(* IEC 61131-3 sources: vertical-injection-machine-docs/docs/IM_SYS_PRG/Code/面板管理/面板公用, 7 files *)

(* ---- PanelTypes.st ---- *)
(*
  PanelTypes.st
  功能：
  1. 定义面板管理层统一使用的按键点位结构和综合按键结构。
  2. 统一收口“面板排序号 + 按键值 + 按键灯”三类信息，避免键值与灯值分散绑定。
  3. 为 `FB_MK110`、`FB_MK116`、`FB_MK150` 提供稳定的数据边界。

  说明：
  1. `uiPanelOrder` 由具体面板功能块按各自型号写入，`0` 表示当前面板未安装该逻辑键位。
  2. `bValue` 由面板输入解码逻辑回写，表示当前逻辑键是否被按下。
  3. `bLamp` 由上层控制逻辑写入，表示当前逻辑键对应的灯是否需要点亮。
*)

TYPE ST_PanelButton :
STRUCT
    uiPanelOrder: UINT;     // 当前逻辑键在当前面板型号中的排序号；`0` 表示该面板型号不提供此键位。
    bValue: BOOL;           // 当前逻辑键输入值；由面板功能块根据输入字和排序号解码后回写。
    bLamp: BOOL;            // 当前逻辑键灯输出请求；由上层写入，再由面板功能块按排序号编码到输出字。
END_STRUCT
END_TYPE

TYPE ST_PanelButtons :
STRUCT
    stManual: ST_PanelButton;            // 手动键综合点位，统一收口其排序号、键值和灯值。
    stSemiautomatic: ST_PanelButton;     // 半自动键综合点位，统一收口其排序号、键值和灯值。
    stAutomatic: ST_PanelButton;         // 全自动键综合点位，统一收口其排序号、键值和灯值。
    stAdjustMold: ST_PanelButton;        // 调模键综合点位，统一收口其排序号、键值和灯值。
    stHeat: ST_PanelButton;              // 电热键综合点位，统一收口其排序号、键值和灯值。
    stMotor: ST_PanelButton;             // 马达键综合点位，统一收口其排序号、键值和灯值。
    stMoldOpen: ST_PanelButton;          // 开模键综合点位，统一收口其排序号、键值和灯值。
    stMoldClose: ST_PanelButton;         // 锁模键综合点位，统一收口其排序号、键值和灯值。
    stMaterialMelt: ST_PanelButton;      // 储料键综合点位，统一收口其排序号、键值和灯值。
    stCleanMaterial: ST_PanelButton;     // 清料键综合点位，统一收口其排序号、键值和灯值。
    stJetLube: ST_PanelButton;           // 润滑键综合点位，统一收口其排序号、键值和灯值。
    stInjFwd: ST_PanelButton;            // 射出键综合点位，统一收口其排序号、键值和灯值。
    stInjBwd: ST_PanelButton;            // 射退键综合点位，统一收口其排序号、键值和灯值。
    stPressRise: ST_PanelButton;         // 压力加键综合点位，统一收口其排序号、键值和灯值。
    stPressFall: ST_PanelButton;         // 压力减键综合点位，统一收口其排序号、键值和灯值。
    stEjectorFwd: ST_PanelButton;        // 托模进键综合点位，统一收口其排序号、键值和灯值。
    stEjectorBwd: ST_PanelButton;        // 托模退键综合点位，统一收口其排序号、键值和灯值。
    stMultiEjector: ST_PanelButton;      // 多次托模键综合点位，统一收口其排序号、键值和灯值。
    stBlow: ST_PanelButton;              // 吹气键综合点位，统一收口其排序号、键值和灯值。
    stInjUnitFwd: ST_PanelButton;        // 座进键综合点位，统一收口其排序号、键值和灯值。
    stInjUnitBwd: ST_PanelButton;        // 座退键综合点位，统一收口其排序号、键值和灯值。
    stLockFwd: ST_PanelButton;           // 定位进键综合点位，统一收口其排序号、键值和灯值。
    stLockBwd: ST_PanelButton;           // 定位退键综合点位，统一收口其排序号、键值和灯值。
    stCoreFwdA: ST_PanelButton;          // 中子 A 进键综合点位，统一收口其排序号、键值和灯值。
    stCoreBwdA: ST_PanelButton;          // 中子 A 退键综合点位，统一收口其排序号、键值和灯值。
    stZipperBwd: ST_PanelButton;         // 倒带键综合点位，统一收口其排序号、键值和灯值。
    stZipperFwd: ST_PanelButton;         // 拉带键综合点位，统一收口其排序号、键值和灯值。
    stZipperClamp: ST_PanelButton;       // 夹带键综合点位，统一收口其排序号、键值和灯值。
    stZipperMotor: ST_PanelButton;       // 拉带马达键综合点位，统一收口其排序号、键值和灯值。
END_STRUCT
END_TYPE

(* ---- F_PanelReadKeyByOrder.st ---- *)
(*
  F_PanelReadKeyByOrder 函数
  功能：
  1. 按统一的面板排序号，从 4 个面板输入字中解码当前逻辑键的实际按键值。
  2. 约定排序号 `1..16` 对应 `uiIN0` 的 `0..15` 位，排序号 `17..32` 对应 `uiIN1` 的 `0..15` 位。
  3. 供 `FB_Panel` 以及各具体面板型号功能块复用，避免每个型号都重复展开读键分支。
*)
FUNCTION F_PanelReadKeyByOrder : BOOL
VAR_INPUT
    uiPanelOrder: UINT;       // 当前待解码的面板排序号；由具体面板功能块按当前型号写入。
    uiIN0: UINT;              // 面板输入字 0；承载排序号 `1..16` 对应的键输入。
    uiIN1: UINT;              // 面板输入字 1；承载排序号 `17..32` 对应的键输入。
    uiIN2: UINT;              // 面板输入字 2；承载排序号 `33..48` 对应的键输入。
    uiIN3: UINT;              // 面板输入字 3；承载排序号 `49..64` 对应的键输入。
END_VAR

IF uiPanelOrder = UINT#0 THEN
    F_PanelReadKeyByOrder := FALSE;                                                             // 排序号为 0 时表示当前面板型号不提供该逻辑键，因此直接回读 FALSE。
ELSIF (uiPanelOrder >= UINT#1) AND (uiPanelOrder <= UINT#16) THEN
    F_PanelReadKeyByOrder := F_PanelGetBit(uiValue := uiIN0, uiBitIndex := uiPanelOrder - UINT#1);   // 排序号落在 `1..16` 时，从 `uiIN0` 的对应位读取当前键值。
ELSIF (uiPanelOrder >= UINT#17) AND (uiPanelOrder <= UINT#32) THEN
    F_PanelReadKeyByOrder := F_PanelGetBit(uiValue := uiIN1, uiBitIndex := uiPanelOrder - UINT#17);  // 排序号落在 `17..32` 时，从 `uiIN1` 的对应位读取当前键值。
ELSIF (uiPanelOrder >= UINT#33) AND (uiPanelOrder <= UINT#48) THEN
    F_PanelReadKeyByOrder := F_PanelGetBit(uiValue := uiIN2, uiBitIndex := uiPanelOrder - UINT#33);  // 排序号落在 `33..48` 时，从 `uiIN2` 的对应位读取当前键值。
ELSIF (uiPanelOrder >= UINT#49) AND (uiPanelOrder <= UINT#64) THEN
    F_PanelReadKeyByOrder := F_PanelGetBit(uiValue := uiIN3, uiBitIndex := uiPanelOrder - UINT#49);  // 排序号落在 `49..64` 时，从 `uiIN3` 的对应位读取当前键值。
ELSE
    F_PanelReadKeyByOrder := FALSE;                                                             // 排序号超出统一支持范围时直接回读 FALSE，避免访问非法位。
END_IF;
END_FUNCTION

(* ---- F_PanelSetBit.st ---- *)
(*
  F_PanelSetBit 函数
  功能：
  1. 按位索引对一个 `UINT` 做置位或清位操作。
  2. 供面板灯输出逻辑按“排序号 -> 输出位”的方式统一生成输出字。
  3. 越界位索引会直接返回原字，避免上层输出字被非法写坏。
*)
FUNCTION F_PanelSetBit : UINT
VAR_INPUT
    uiValue: UINT;         // 待修改的目标字；通常来自面板输出字 `uiOUT0` 或 `uiOUT1`。
    uiBitIndex: UINT;      // 目标位索引；有效范围为 `0..15`。
    bBitValue: BOOL;       // TRUE=把目标位置 1；FALSE=把目标位清 0。
END_VAR

IF uiBitIndex > 15 THEN
    F_PanelSetBit := uiValue;                                                     // 位索引越界时保持原字不变，避免误改无关输出位。
ELSIF bBitValue THEN
    F_PanelSetBit := uiValue OR SHL(UINT#1, uiBitIndex);                          // 需要点亮时，用位掩码把目标位置 1。
ELSE
    F_PanelSetBit := uiValue AND NOT SHL(UINT#1, uiBitIndex);                     // 需要熄灭时，用位掩码把目标位清 0。
END_IF;
END_FUNCTION

(* ---- FB_Panel.st ---- *)
(*
  FB_Panel 功能块
  功能：
  1. 统一按 `stPanelButtons.*.uiPanelOrder` 完成全部逻辑键的输入解码和灯输出编码。
  2. 让各具体面板型号功能块只负责定义当前型号的排序号，不需要再重复展开整块读键/写灯流程。
  3. 当前块本体不关心具体型号是 MK110、MK116 还是 MK150，只按排序号执行。
*)
FUNCTION_BLOCK FB_Panel
VAR_IN_OUT
    stPanelButtons: ST_PanelButtons;     // 综合面板按键结构；调用方先写入排序号和灯值，本块再回写键值并生成灯输出。
END_VAR
VAR_INPUT
    uiIN0: UINT;                         // 面板输入字 0；承载排序号 `1..16` 对应的键输入。
    uiIN1: UINT;                         // 面板输入字 1；承载排序号 `17..32` 对应的键输入。
    uiIN2: UINT;                         // 面板输入字 2；承载排序号 `33..48` 对应的键输入。
    uiIN3: UINT;                         // 面板输入字 3；承载排序号 `49..64` 对应的键输入。
END_VAR
VAR_OUTPUT
    uiOUT0: UINT;                        // 面板输出字 0；承载排序号 `1..16` 对应的灯输出。
    uiOUT1: UINT;                        // 面板输出字 1；承载排序号 `17..32` 对应的灯输出。
    uiOUT2: UINT;                        // 面板输出字 2；承载排序号 `33..48` 对应的灯输出。
    uiOUT3: UINT;                        // 面板输出字 3；承载排序号 `49..64` 对应的灯输出。
END_VAR
VAR
    fbLampWriter: FB_PanelLampWriter;    // 通用面板灯写入器；负责把单个逻辑键的灯请求并入统一输出字。
END_VAR

(* 先统一按排序号解码全部逻辑键的当前输入值。 *)
stPanelButtons.stManual.bValue := F_PanelReadKeyByOrder(uiPanelOrder := stPanelButtons.stManual.uiPanelOrder, uiIN0 := uiIN0, uiIN1 := uiIN1, uiIN2 := uiIN2, uiIN3 := uiIN3);                         // 读取手动键当前值。
stPanelButtons.stSemiautomatic.bValue := F_PanelReadKeyByOrder(uiPanelOrder := stPanelButtons.stSemiautomatic.uiPanelOrder, uiIN0 := uiIN0, uiIN1 := uiIN1, uiIN2 := uiIN2, uiIN3 := uiIN3);          // 读取半自动键当前值。
stPanelButtons.stAutomatic.bValue := F_PanelReadKeyByOrder(uiPanelOrder := stPanelButtons.stAutomatic.uiPanelOrder, uiIN0 := uiIN0, uiIN1 := uiIN1, uiIN2 := uiIN2, uiIN3 := uiIN3);                  // 读取全自动键当前值。
stPanelButtons.stAdjustMold.bValue := F_PanelReadKeyByOrder(uiPanelOrder := stPanelButtons.stAdjustMold.uiPanelOrder, uiIN0 := uiIN0, uiIN1 := uiIN1, uiIN2 := uiIN2, uiIN3 := uiIN3);                // 读取调模键当前值。
stPanelButtons.stHeat.bValue := F_PanelReadKeyByOrder(uiPanelOrder := stPanelButtons.stHeat.uiPanelOrder, uiIN0 := uiIN0, uiIN1 := uiIN1, uiIN2 := uiIN2, uiIN3 := uiIN3);                               // 读取电热键当前值。
stPanelButtons.stMotor.bValue := F_PanelReadKeyByOrder(uiPanelOrder := stPanelButtons.stMotor.uiPanelOrder, uiIN0 := uiIN0, uiIN1 := uiIN1, uiIN2 := uiIN2, uiIN3 := uiIN3);                            // 读取马达键当前值。
stPanelButtons.stMoldOpen.bValue := F_PanelReadKeyByOrder(uiPanelOrder := stPanelButtons.stMoldOpen.uiPanelOrder, uiIN0 := uiIN0, uiIN1 := uiIN1, uiIN2 := uiIN2, uiIN3 := uiIN3);                      // 读取开模键当前值。
stPanelButtons.stMoldClose.bValue := F_PanelReadKeyByOrder(uiPanelOrder := stPanelButtons.stMoldClose.uiPanelOrder, uiIN0 := uiIN0, uiIN1 := uiIN1, uiIN2 := uiIN2, uiIN3 := uiIN3);                    // 读取锁模键当前值。
stPanelButtons.stMaterialMelt.bValue := F_PanelReadKeyByOrder(uiPanelOrder := stPanelButtons.stMaterialMelt.uiPanelOrder, uiIN0 := uiIN0, uiIN1 := uiIN1, uiIN2 := uiIN2, uiIN3 := uiIN3);              // 读取储料键当前值。
stPanelButtons.stCleanMaterial.bValue := F_PanelReadKeyByOrder(uiPanelOrder := stPanelButtons.stCleanMaterial.uiPanelOrder, uiIN0 := uiIN0, uiIN1 := uiIN1, uiIN2 := uiIN2, uiIN3 := uiIN3);            // 读取清料键当前值。
stPanelButtons.stJetLube.bValue := F_PanelReadKeyByOrder(uiPanelOrder := stPanelButtons.stJetLube.uiPanelOrder, uiIN0 := uiIN0, uiIN1 := uiIN1, uiIN2 := uiIN2, uiIN3 := uiIN3);                         // 读取润滑键当前值。
stPanelButtons.stInjFwd.bValue := F_PanelReadKeyByOrder(uiPanelOrder := stPanelButtons.stInjFwd.uiPanelOrder, uiIN0 := uiIN0, uiIN1 := uiIN1, uiIN2 := uiIN2, uiIN3 := uiIN3);                           // 读取射出键当前值。
stPanelButtons.stInjBwd.bValue := F_PanelReadKeyByOrder(uiPanelOrder := stPanelButtons.stInjBwd.uiPanelOrder, uiIN0 := uiIN0, uiIN1 := uiIN1, uiIN2 := uiIN2, uiIN3 := uiIN3);                           // 读取射退键当前值。
stPanelButtons.stPressRise.bValue := F_PanelReadKeyByOrder(uiPanelOrder := stPanelButtons.stPressRise.uiPanelOrder, uiIN0 := uiIN0, uiIN1 := uiIN1, uiIN2 := uiIN2, uiIN3 := uiIN3);                      // 读取压力加键当前值。
stPanelButtons.stPressFall.bValue := F_PanelReadKeyByOrder(uiPanelOrder := stPanelButtons.stPressFall.uiPanelOrder, uiIN0 := uiIN0, uiIN1 := uiIN1, uiIN2 := uiIN2, uiIN3 := uiIN3);                      // 读取压力减键当前值。
stPanelButtons.stEjectorFwd.bValue := F_PanelReadKeyByOrder(uiPanelOrder := stPanelButtons.stEjectorFwd.uiPanelOrder, uiIN0 := uiIN0, uiIN1 := uiIN1, uiIN2 := uiIN2, uiIN3 := uiIN3);                    // 读取托模进键当前值。
stPanelButtons.stEjectorBwd.bValue := F_PanelReadKeyByOrder(uiPanelOrder := stPanelButtons.stEjectorBwd.uiPanelOrder, uiIN0 := uiIN0, uiIN1 := uiIN1, uiIN2 := uiIN2, uiIN3 := uiIN3);                    // 读取托模退键当前值。
stPanelButtons.stMultiEjector.bValue := F_PanelReadKeyByOrder(uiPanelOrder := stPanelButtons.stMultiEjector.uiPanelOrder, uiIN0 := uiIN0, uiIN1 := uiIN1, uiIN2 := uiIN2, uiIN3 := uiIN3);                // 读取多次托模键当前值。
stPanelButtons.stBlow.bValue := F_PanelReadKeyByOrder(uiPanelOrder := stPanelButtons.stBlow.uiPanelOrder, uiIN0 := uiIN0, uiIN1 := uiIN1, uiIN2 := uiIN2, uiIN3 := uiIN3);                               // 读取吹气键当前值。
stPanelButtons.stInjUnitFwd.bValue := F_PanelReadKeyByOrder(uiPanelOrder := stPanelButtons.stInjUnitFwd.uiPanelOrder, uiIN0 := uiIN0, uiIN1 := uiIN1, uiIN2 := uiIN2, uiIN3 := uiIN3);                    // 读取座进键当前值。
stPanelButtons.stInjUnitBwd.bValue := F_PanelReadKeyByOrder(uiPanelOrder := stPanelButtons.stInjUnitBwd.uiPanelOrder, uiIN0 := uiIN0, uiIN1 := uiIN1, uiIN2 := uiIN2, uiIN3 := uiIN3);                    // 读取座退键当前值。
stPanelButtons.stLockFwd.bValue := F_PanelReadKeyByOrder(uiPanelOrder := stPanelButtons.stLockFwd.uiPanelOrder, uiIN0 := uiIN0, uiIN1 := uiIN1, uiIN2 := uiIN2, uiIN3 := uiIN3);                          // 读取定位进键当前值。
stPanelButtons.stLockBwd.bValue := F_PanelReadKeyByOrder(uiPanelOrder := stPanelButtons.stLockBwd.uiPanelOrder, uiIN0 := uiIN0, uiIN1 := uiIN1, uiIN2 := uiIN2, uiIN3 := uiIN3);                          // 读取定位退键当前值。
stPanelButtons.stCoreFwdA.bValue := F_PanelReadKeyByOrder(uiPanelOrder := stPanelButtons.stCoreFwdA.uiPanelOrder, uiIN0 := uiIN0, uiIN1 := uiIN1, uiIN2 := uiIN2, uiIN3 := uiIN3);                        // 读取中子 A 进键当前值。
stPanelButtons.stCoreBwdA.bValue := F_PanelReadKeyByOrder(uiPanelOrder := stPanelButtons.stCoreBwdA.uiPanelOrder, uiIN0 := uiIN0, uiIN1 := uiIN1, uiIN2 := uiIN2, uiIN3 := uiIN3);                        // 读取中子 A 退键当前值。
stPanelButtons.stZipperBwd.bValue := F_PanelReadKeyByOrder(uiPanelOrder := stPanelButtons.stZipperBwd.uiPanelOrder, uiIN0 := uiIN0, uiIN1 := uiIN1, uiIN2 := uiIN2, uiIN3 := uiIN3);                      // 读取倒带键当前值。
stPanelButtons.stZipperFwd.bValue := F_PanelReadKeyByOrder(uiPanelOrder := stPanelButtons.stZipperFwd.uiPanelOrder, uiIN0 := uiIN0, uiIN1 := uiIN1, uiIN2 := uiIN2, uiIN3 := uiIN3);                      // 读取拉带键当前值。
stPanelButtons.stZipperClamp.bValue := F_PanelReadKeyByOrder(uiPanelOrder := stPanelButtons.stZipperClamp.uiPanelOrder, uiIN0 := uiIN0, uiIN1 := uiIN1, uiIN2 := uiIN2, uiIN3 := uiIN3);                  // 读取夹带键当前值。
stPanelButtons.stZipperMotor.bValue := F_PanelReadKeyByOrder(uiPanelOrder := stPanelButtons.stZipperMotor.uiPanelOrder, uiIN0 := uiIN0, uiIN1 := uiIN1, uiIN2 := uiIN2, uiIN3 := uiIN3);                  // 读取拉带马达键当前值。

(* 再先清零 4 个统一输出字，准备在本扫描周期重新汇总灯输出。 *)
uiOUT0 := UINT#0;                        // 清零输出字 0，避免上一拍残留的灯位继续保留。
uiOUT1 := UINT#0;                        // 清零输出字 1，避免上一拍残留的灯位继续保留。
uiOUT2 := UINT#0;                        // 清零输出字 2，避免上一拍残留的灯位继续保留。
uiOUT3 := UINT#0;                        // 清零输出字 3，避免上一拍残留的灯位继续保留。

(* 最后按同一排序号统一生成灯输出。 *)
fbLampWriter(uiOUT0 := uiOUT0, uiOUT1 := uiOUT1, uiOUT2 := uiOUT2, uiOUT3 := uiOUT3, uiPanelOrder := stPanelButtons.stManual.uiPanelOrder, bLampValue := stPanelButtons.stManual.bLamp);                        // 并入手动键灯请求。
fbLampWriter(uiOUT0 := uiOUT0, uiOUT1 := uiOUT1, uiOUT2 := uiOUT2, uiOUT3 := uiOUT3, uiPanelOrder := stPanelButtons.stSemiautomatic.uiPanelOrder, bLampValue := stPanelButtons.stSemiautomatic.bLamp);        // 并入半自动键灯请求。
fbLampWriter(uiOUT0 := uiOUT0, uiOUT1 := uiOUT1, uiOUT2 := uiOUT2, uiOUT3 := uiOUT3, uiPanelOrder := stPanelButtons.stAutomatic.uiPanelOrder, bLampValue := stPanelButtons.stAutomatic.bLamp);                 // 并入全自动键灯请求。
fbLampWriter(uiOUT0 := uiOUT0, uiOUT1 := uiOUT1, uiOUT2 := uiOUT2, uiOUT3 := uiOUT3, uiPanelOrder := stPanelButtons.stAdjustMold.uiPanelOrder, bLampValue := stPanelButtons.stAdjustMold.bLamp);              // 并入调模键灯请求。
fbLampWriter(uiOUT0 := uiOUT0, uiOUT1 := uiOUT1, uiOUT2 := uiOUT2, uiOUT3 := uiOUT3, uiPanelOrder := stPanelButtons.stHeat.uiPanelOrder, bLampValue := stPanelButtons.stHeat.bLamp);                           // 并入电热键灯请求。
fbLampWriter(uiOUT0 := uiOUT0, uiOUT1 := uiOUT1, uiOUT2 := uiOUT2, uiOUT3 := uiOUT3, uiPanelOrder := stPanelButtons.stMotor.uiPanelOrder, bLampValue := stPanelButtons.stMotor.bLamp);                         // 并入马达键灯请求。
fbLampWriter(uiOUT0 := uiOUT0, uiOUT1 := uiOUT1, uiOUT2 := uiOUT2, uiOUT3 := uiOUT3, uiPanelOrder := stPanelButtons.stMoldOpen.uiPanelOrder, bLampValue := stPanelButtons.stMoldOpen.bLamp);                  // 并入开模键灯请求。
fbLampWriter(uiOUT0 := uiOUT0, uiOUT1 := uiOUT1, uiOUT2 := uiOUT2, uiOUT3 := uiOUT3, uiPanelOrder := stPanelButtons.stMoldClose.uiPanelOrder, bLampValue := stPanelButtons.stMoldClose.bLamp);                // 并入锁模键灯请求。
fbLampWriter(uiOUT0 := uiOUT0, uiOUT1 := uiOUT1, uiOUT2 := uiOUT2, uiOUT3 := uiOUT3, uiPanelOrder := stPanelButtons.stMaterialMelt.uiPanelOrder, bLampValue := stPanelButtons.stMaterialMelt.bLamp);          // 并入储料键灯请求。
fbLampWriter(uiOUT0 := uiOUT0, uiOUT1 := uiOUT1, uiOUT2 := uiOUT2, uiOUT3 := uiOUT3, uiPanelOrder := stPanelButtons.stCleanMaterial.uiPanelOrder, bLampValue := stPanelButtons.stCleanMaterial.bLamp);        // 并入清料键灯请求。
fbLampWriter(uiOUT0 := uiOUT0, uiOUT1 := uiOUT1, uiOUT2 := uiOUT2, uiOUT3 := uiOUT3, uiPanelOrder := stPanelButtons.stJetLube.uiPanelOrder, bLampValue := stPanelButtons.stJetLube.bLamp);                    // 并入润滑键灯请求。
fbLampWriter(uiOUT0 := uiOUT0, uiOUT1 := uiOUT1, uiOUT2 := uiOUT2, uiOUT3 := uiOUT3, uiPanelOrder := stPanelButtons.stInjFwd.uiPanelOrder, bLampValue := stPanelButtons.stInjFwd.bLamp);                       // 并入射出键灯请求。
fbLampWriter(uiOUT0 := uiOUT0, uiOUT1 := uiOUT1, uiOUT2 := uiOUT2, uiOUT3 := uiOUT3, uiPanelOrder := stPanelButtons.stInjBwd.uiPanelOrder, bLampValue := stPanelButtons.stInjBwd.bLamp);                       // 并入射退键灯请求。
fbLampWriter(uiOUT0 := uiOUT0, uiOUT1 := uiOUT1, uiOUT2 := uiOUT2, uiOUT3 := uiOUT3, uiPanelOrder := stPanelButtons.stPressRise.uiPanelOrder, bLampValue := stPanelButtons.stPressRise.bLamp);                // 并入压力加键灯请求。
fbLampWriter(uiOUT0 := uiOUT0, uiOUT1 := uiOUT1, uiOUT2 := uiOUT2, uiOUT3 := uiOUT3, uiPanelOrder := stPanelButtons.stPressFall.uiPanelOrder, bLampValue := stPanelButtons.stPressFall.bLamp);                // 并入压力减键灯请求。
fbLampWriter(uiOUT0 := uiOUT0, uiOUT1 := uiOUT1, uiOUT2 := uiOUT2, uiOUT3 := uiOUT3, uiPanelOrder := stPanelButtons.stEjectorFwd.uiPanelOrder, bLampValue := stPanelButtons.stEjectorFwd.bLamp);              // 并入托模进键灯请求。
fbLampWriter(uiOUT0 := uiOUT0, uiOUT1 := uiOUT1, uiOUT2 := uiOUT2, uiOUT3 := uiOUT3, uiPanelOrder := stPanelButtons.stEjectorBwd.uiPanelOrder, bLampValue := stPanelButtons.stEjectorBwd.bLamp);              // 并入托模退键灯请求。
fbLampWriter(uiOUT0 := uiOUT0, uiOUT1 := uiOUT1, uiOUT2 := uiOUT2, uiOUT3 := uiOUT3, uiPanelOrder := stPanelButtons.stMultiEjector.uiPanelOrder, bLampValue := stPanelButtons.stMultiEjector.bLamp);          // 并入多次托模键灯请求。
fbLampWriter(uiOUT0 := uiOUT0, uiOUT1 := uiOUT1, uiOUT2 := uiOUT2, uiOUT3 := uiOUT3, uiPanelOrder := stPanelButtons.stBlow.uiPanelOrder, bLampValue := stPanelButtons.stBlow.bLamp);                           // 并入吹气键灯请求。
fbLampWriter(uiOUT0 := uiOUT0, uiOUT1 := uiOUT1, uiOUT2 := uiOUT2, uiOUT3 := uiOUT3, uiPanelOrder := stPanelButtons.stInjUnitFwd.uiPanelOrder, bLampValue := stPanelButtons.stInjUnitFwd.bLamp);              // 并入座进键灯请求。
fbLampWriter(uiOUT0 := uiOUT0, uiOUT1 := uiOUT1, uiOUT2 := uiOUT2, uiOUT3 := uiOUT3, uiPanelOrder := stPanelButtons.stInjUnitBwd.uiPanelOrder, bLampValue := stPanelButtons.stInjUnitBwd.bLamp);              // 并入座退键灯请求。
fbLampWriter(uiOUT0 := uiOUT0, uiOUT1 := uiOUT1, uiOUT2 := uiOUT2, uiOUT3 := uiOUT3, uiPanelOrder := stPanelButtons.stLockFwd.uiPanelOrder, bLampValue := stPanelButtons.stLockFwd.bLamp);                   // 并入定位进键灯请求。
fbLampWriter(uiOUT0 := uiOUT0, uiOUT1 := uiOUT1, uiOUT2 := uiOUT2, uiOUT3 := uiOUT3, uiPanelOrder := stPanelButtons.stLockBwd.uiPanelOrder, bLampValue := stPanelButtons.stLockBwd.bLamp);                   // 并入定位退键灯请求。
fbLampWriter(uiOUT0 := uiOUT0, uiOUT1 := uiOUT1, uiOUT2 := uiOUT2, uiOUT3 := uiOUT3, uiPanelOrder := stPanelButtons.stCoreFwdA.uiPanelOrder, bLampValue := stPanelButtons.stCoreFwdA.bLamp);                // 并入中子 A 进键灯请求。
fbLampWriter(uiOUT0 := uiOUT0, uiOUT1 := uiOUT1, uiOUT2 := uiOUT2, uiOUT3 := uiOUT3, uiPanelOrder := stPanelButtons.stCoreBwdA.uiPanelOrder, bLampValue := stPanelButtons.stCoreBwdA.bLamp);                // 并入中子 A 退键灯请求。
fbLampWriter(uiOUT0 := uiOUT0, uiOUT1 := uiOUT1, uiOUT2 := uiOUT2, uiOUT3 := uiOUT3, uiPanelOrder := stPanelButtons.stZipperBwd.uiPanelOrder, bLampValue := stPanelButtons.stZipperBwd.bLamp);              // 并入倒带键灯请求。
fbLampWriter(uiOUT0 := uiOUT0, uiOUT1 := uiOUT1, uiOUT2 := uiOUT2, uiOUT3 := uiOUT3, uiPanelOrder := stPanelButtons.stZipperFwd.uiPanelOrder, bLampValue := stPanelButtons.stZipperFwd.bLamp);              // 并入拉带键灯请求。
fbLampWriter(uiOUT0 := uiOUT0, uiOUT1 := uiOUT1, uiOUT2 := uiOUT2, uiOUT3 := uiOUT3, uiPanelOrder := stPanelButtons.stZipperClamp.uiPanelOrder, bLampValue := stPanelButtons.stZipperClamp.bLamp);            // 并入夹带键灯请求。
fbLampWriter(uiOUT0 := uiOUT0, uiOUT1 := uiOUT1, uiOUT2 := uiOUT2, uiOUT3 := uiOUT3, uiPanelOrder := stPanelButtons.stZipperMotor.uiPanelOrder, bLampValue := stPanelButtons.stZipperMotor.bLamp);            // 并入拉带马达键灯请求。
END_FUNCTION_BLOCK

(* ---- FB_PanelLampEncoder.st ---- *)
(*
  FB_PanelLampEncoder 功能块
  功能：
  1. 统一按 `stPanelButtons.*.uiPanelOrder` 把全部逻辑灯请求编码到 `uiOUT0..uiOUT3`。
  2. 让具体面板型号块与面板调度块只维护灯请求，不再重复展开整块写灯逻辑。
  3. 当前块只处理“写灯”，不负责读取按键值。
*)
FUNCTION_BLOCK FB_PanelLampEncoder
VAR_INPUT
    stPanelButtons: ST_PanelButtons;     // 综合面板按键结构；本块读取其中全部逻辑键灯请求与排序号来生成输出字。
END_VAR
VAR_OUTPUT
    uiOUT0: UINT;                        // 面板输出字 0；按 `uiPanelOrder` 汇总排序号 `1..16` 的灯输出。
    uiOUT1: UINT;                        // 面板输出字 1；按 `uiPanelOrder` 汇总排序号 `17..32` 的灯输出。
    uiOUT2: UINT;                        // 面板输出字 2；按 `uiPanelOrder` 汇总排序号 `33..48` 的灯输出。
    uiOUT3: UINT;                        // 面板输出字 3；按 `uiPanelOrder` 汇总排序号 `49..64` 的灯输出。
END_VAR
VAR
    fbLampWriter: FB_PanelLampWriter;    // 通用面板灯写入器；负责把单个逻辑键的灯请求并入统一输出字。
END_VAR

uiOUT0 := UINT#0;                        // 每拍先清零输出字 0，避免上一拍残留的灯位继续保留。
uiOUT1 := UINT#0;                        // 每拍先清零输出字 1，避免上一拍残留的灯位继续保留。
uiOUT2 := UINT#0;                        // 每拍先清零输出字 2，避免上一拍残留的灯位继续保留。
uiOUT3 := UINT#0;                        // 每拍先清零输出字 3，避免上一拍残留的灯位继续保留。

fbLampWriter(uiOUT0 := uiOUT0, uiOUT1 := uiOUT1, uiOUT2 := uiOUT2, uiOUT3 := uiOUT3, uiPanelOrder := stPanelButtons.stManual.uiPanelOrder, bLampValue := stPanelButtons.stManual.bLamp);                        // 并入手动键灯请求。
fbLampWriter(uiOUT0 := uiOUT0, uiOUT1 := uiOUT1, uiOUT2 := uiOUT2, uiOUT3 := uiOUT3, uiPanelOrder := stPanelButtons.stSemiautomatic.uiPanelOrder, bLampValue := stPanelButtons.stSemiautomatic.bLamp);        // 并入半自动键灯请求。
fbLampWriter(uiOUT0 := uiOUT0, uiOUT1 := uiOUT1, uiOUT2 := uiOUT2, uiOUT3 := uiOUT3, uiPanelOrder := stPanelButtons.stAutomatic.uiPanelOrder, bLampValue := stPanelButtons.stAutomatic.bLamp);                 // 并入全自动键灯请求。
fbLampWriter(uiOUT0 := uiOUT0, uiOUT1 := uiOUT1, uiOUT2 := uiOUT2, uiOUT3 := uiOUT3, uiPanelOrder := stPanelButtons.stAdjustMold.uiPanelOrder, bLampValue := stPanelButtons.stAdjustMold.bLamp);              // 并入调模键灯请求。
fbLampWriter(uiOUT0 := uiOUT0, uiOUT1 := uiOUT1, uiOUT2 := uiOUT2, uiOUT3 := uiOUT3, uiPanelOrder := stPanelButtons.stHeat.uiPanelOrder, bLampValue := stPanelButtons.stHeat.bLamp);                           // 并入电热键灯请求。
fbLampWriter(uiOUT0 := uiOUT0, uiOUT1 := uiOUT1, uiOUT2 := uiOUT2, uiOUT3 := uiOUT3, uiPanelOrder := stPanelButtons.stMotor.uiPanelOrder, bLampValue := stPanelButtons.stMotor.bLamp);                         // 并入马达键灯请求。
fbLampWriter(uiOUT0 := uiOUT0, uiOUT1 := uiOUT1, uiOUT2 := uiOUT2, uiOUT3 := uiOUT3, uiPanelOrder := stPanelButtons.stMoldOpen.uiPanelOrder, bLampValue := stPanelButtons.stMoldOpen.bLamp);                  // 并入开模键灯请求。
fbLampWriter(uiOUT0 := uiOUT0, uiOUT1 := uiOUT1, uiOUT2 := uiOUT2, uiOUT3 := uiOUT3, uiPanelOrder := stPanelButtons.stMoldClose.uiPanelOrder, bLampValue := stPanelButtons.stMoldClose.bLamp);                // 并入锁模键灯请求。
fbLampWriter(uiOUT0 := uiOUT0, uiOUT1 := uiOUT1, uiOUT2 := uiOUT2, uiOUT3 := uiOUT3, uiPanelOrder := stPanelButtons.stMaterialMelt.uiPanelOrder, bLampValue := stPanelButtons.stMaterialMelt.bLamp);          // 并入储料键灯请求。
fbLampWriter(uiOUT0 := uiOUT0, uiOUT1 := uiOUT1, uiOUT2 := uiOUT2, uiOUT3 := uiOUT3, uiPanelOrder := stPanelButtons.stCleanMaterial.uiPanelOrder, bLampValue := stPanelButtons.stCleanMaterial.bLamp);        // 并入清料键灯请求。
fbLampWriter(uiOUT0 := uiOUT0, uiOUT1 := uiOUT1, uiOUT2 := uiOUT2, uiOUT3 := uiOUT3, uiPanelOrder := stPanelButtons.stJetLube.uiPanelOrder, bLampValue := stPanelButtons.stJetLube.bLamp);                    // 并入润滑键灯请求。
fbLampWriter(uiOUT0 := uiOUT0, uiOUT1 := uiOUT1, uiOUT2 := uiOUT2, uiOUT3 := uiOUT3, uiPanelOrder := stPanelButtons.stInjFwd.uiPanelOrder, bLampValue := stPanelButtons.stInjFwd.bLamp);                       // 并入射出键灯请求。
fbLampWriter(uiOUT0 := uiOUT0, uiOUT1 := uiOUT1, uiOUT2 := uiOUT2, uiOUT3 := uiOUT3, uiPanelOrder := stPanelButtons.stInjBwd.uiPanelOrder, bLampValue := stPanelButtons.stInjBwd.bLamp);                       // 并入射退键灯请求。
fbLampWriter(uiOUT0 := uiOUT0, uiOUT1 := uiOUT1, uiOUT2 := uiOUT2, uiOUT3 := uiOUT3, uiPanelOrder := stPanelButtons.stPressRise.uiPanelOrder, bLampValue := stPanelButtons.stPressRise.bLamp);                // 并入压力加键灯请求。
fbLampWriter(uiOUT0 := uiOUT0, uiOUT1 := uiOUT1, uiOUT2 := uiOUT2, uiOUT3 := uiOUT3, uiPanelOrder := stPanelButtons.stPressFall.uiPanelOrder, bLampValue := stPanelButtons.stPressFall.bLamp);                // 并入压力减键灯请求。
fbLampWriter(uiOUT0 := uiOUT0, uiOUT1 := uiOUT1, uiOUT2 := uiOUT2, uiOUT3 := uiOUT3, uiPanelOrder := stPanelButtons.stEjectorFwd.uiPanelOrder, bLampValue := stPanelButtons.stEjectorFwd.bLamp);              // 并入托模进键灯请求。
fbLampWriter(uiOUT0 := uiOUT0, uiOUT1 := uiOUT1, uiOUT2 := uiOUT2, uiOUT3 := uiOUT3, uiPanelOrder := stPanelButtons.stEjectorBwd.uiPanelOrder, bLampValue := stPanelButtons.stEjectorBwd.bLamp);              // 并入托模退键灯请求。
fbLampWriter(uiOUT0 := uiOUT0, uiOUT1 := uiOUT1, uiOUT2 := uiOUT2, uiOUT3 := uiOUT3, uiPanelOrder := stPanelButtons.stMultiEjector.uiPanelOrder, bLampValue := stPanelButtons.stMultiEjector.bLamp);          // 并入多次托模键灯请求。
fbLampWriter(uiOUT0 := uiOUT0, uiOUT1 := uiOUT1, uiOUT2 := uiOUT2, uiOUT3 := uiOUT3, uiPanelOrder := stPanelButtons.stBlow.uiPanelOrder, bLampValue := stPanelButtons.stBlow.bLamp);                           // 并入吹气键灯请求。
fbLampWriter(uiOUT0 := uiOUT0, uiOUT1 := uiOUT1, uiOUT2 := uiOUT2, uiOUT3 := uiOUT3, uiPanelOrder := stPanelButtons.stInjUnitFwd.uiPanelOrder, bLampValue := stPanelButtons.stInjUnitFwd.bLamp);              // 并入座进键灯请求。
fbLampWriter(uiOUT0 := uiOUT0, uiOUT1 := uiOUT1, uiOUT2 := uiOUT2, uiOUT3 := uiOUT3, uiPanelOrder := stPanelButtons.stInjUnitBwd.uiPanelOrder, bLampValue := stPanelButtons.stInjUnitBwd.bLamp);              // 并入座退键灯请求。
fbLampWriter(uiOUT0 := uiOUT0, uiOUT1 := uiOUT1, uiOUT2 := uiOUT2, uiOUT3 := uiOUT3, uiPanelOrder := stPanelButtons.stLockFwd.uiPanelOrder, bLampValue := stPanelButtons.stLockFwd.bLamp);                   // 并入定位进键灯请求。
fbLampWriter(uiOUT0 := uiOUT0, uiOUT1 := uiOUT1, uiOUT2 := uiOUT2, uiOUT3 := uiOUT3, uiPanelOrder := stPanelButtons.stLockBwd.uiPanelOrder, bLampValue := stPanelButtons.stLockBwd.bLamp);                   // 并入定位退键灯请求。
fbLampWriter(uiOUT0 := uiOUT0, uiOUT1 := uiOUT1, uiOUT2 := uiOUT2, uiOUT3 := uiOUT3, uiPanelOrder := stPanelButtons.stCoreFwdA.uiPanelOrder, bLampValue := stPanelButtons.stCoreFwdA.bLamp);                // 并入中子 A 进键灯请求。
fbLampWriter(uiOUT0 := uiOUT0, uiOUT1 := uiOUT1, uiOUT2 := uiOUT2, uiOUT3 := uiOUT3, uiPanelOrder := stPanelButtons.stCoreBwdA.uiPanelOrder, bLampValue := stPanelButtons.stCoreBwdA.bLamp);                // 并入中子 A 退键灯请求。
fbLampWriter(uiOUT0 := uiOUT0, uiOUT1 := uiOUT1, uiOUT2 := uiOUT2, uiOUT3 := uiOUT3, uiPanelOrder := stPanelButtons.stZipperBwd.uiPanelOrder, bLampValue := stPanelButtons.stZipperBwd.bLamp);              // 并入倒带键灯请求。
fbLampWriter(uiOUT0 := uiOUT0, uiOUT1 := uiOUT1, uiOUT2 := uiOUT2, uiOUT3 := uiOUT3, uiPanelOrder := stPanelButtons.stZipperFwd.uiPanelOrder, bLampValue := stPanelButtons.stZipperFwd.bLamp);              // 并入拉带键灯请求。
fbLampWriter(uiOUT0 := uiOUT0, uiOUT1 := uiOUT1, uiOUT2 := uiOUT2, uiOUT3 := uiOUT3, uiPanelOrder := stPanelButtons.stZipperClamp.uiPanelOrder, bLampValue := stPanelButtons.stZipperClamp.bLamp);            // 并入夹带键灯请求。
fbLampWriter(uiOUT0 := uiOUT0, uiOUT1 := uiOUT1, uiOUT2 := uiOUT2, uiOUT3 := uiOUT3, uiPanelOrder := stPanelButtons.stZipperMotor.uiPanelOrder, bLampValue := stPanelButtons.stZipperMotor.bLamp);            // 并入拉带马达键灯请求。
END_FUNCTION_BLOCK

(* ---- FB_PanelLampWriter.st ---- *)
(*
  FB_PanelLampWriter 功能块
  功能：
  1. 按统一的面板排序号，把单个逻辑键的灯请求写入 `uiOUT0/uiOUT1`。
  2. 约定排序号 `1..16` 对应 `uiOUT0` 的 `0..15` 位，排序号 `17..32` 对应 `uiOUT1` 的 `0..15` 位。
  3. 供 `FB_MK110`、`FB_MK116`、`FB_MK150` 复用，避免每个面板块重复展开灯位写入分支。

  使用约束：
  1. 调用方必须在本扫描周期开始前先把 `uiOUT0`、`uiOUT1` 清零。
  2. 本块只负责把单个逻辑键的灯请求并入输出字，不负责排序号唯一性检查。
*)
FUNCTION_BLOCK FB_PanelLampWriter
VAR_IN_OUT
    uiOUT0: UINT;             // 输出字 0；承载排序号 `1..16` 对应的面板灯位。
    uiOUT1: UINT;             // 输出字 1；承载排序号 `17..32` 对应的面板灯位。
    uiOUT2: UINT;             // 输出字 2；承载排序号 `33..48` 对应的面板灯位。
    uiOUT3: UINT;             // 输出字 3；承载排序号 `49..64` 对应的面板灯位。
END_VAR
VAR_INPUT
    uiPanelOrder: UINT;       // 当前逻辑键在当前面板型号中的排序号；`0` 表示本次不写任何灯位。
    bLampValue: BOOL;         // 当前逻辑键的灯请求；TRUE=点亮对应灯位，FALSE=保持输出字当前值不变。
END_VAR

IF NOT bLampValue THEN
    (* 当前逻辑键灯请求为 FALSE 时不做任何写入。
       调用方已在扫描周期开始时统一清零输出字，因此这里不需要再重复清位。
    *)
ELSIF (uiPanelOrder >= 1) AND (uiPanelOrder <= 16) THEN
    uiOUT0 := F_PanelSetBit(uiValue := uiOUT0, uiBitIndex := uiPanelOrder - 1, bBitValue := TRUE);   // 排序号落在 `1..16` 时，把灯写入 `uiOUT0` 的对应位。
ELSIF (uiPanelOrder >= 17) AND (uiPanelOrder <= 32) THEN
    uiOUT1 := F_PanelSetBit(uiValue := uiOUT1, uiBitIndex := uiPanelOrder - 17, bBitValue := TRUE);  // 排序号落在 `17..32` 时，把灯写入 `uiOUT1` 的对应位。
ELSIF (uiPanelOrder >= 33) AND (uiPanelOrder <= 48) THEN
    uiOUT2 := F_PanelSetBit(uiValue := uiOUT2, uiBitIndex := uiPanelOrder - 33, bBitValue := TRUE);  // 排序号落在 `33..48` 时，把灯写入 `uiOUT2` 的对应位。
ELSIF (uiPanelOrder >= 49) AND (uiPanelOrder <= 64) THEN
    uiOUT3 := F_PanelSetBit(uiValue := uiOUT3, uiBitIndex := uiPanelOrder - 49, bBitValue := TRUE);  // 排序号落在 `49..64` 时，把灯写入 `uiOUT3` 的对应位。
END_IF;
END_FUNCTION_BLOCK

(* ---- FB_PanelReader.st ---- *)
(*
  FB_PanelReader 功能块
  功能：
  1. 统一按 `stPanelButtons.*` 中保存的真实输入字号与位号回写全部逻辑键当前值。
  2. 让具体面板型号块只负责维护映射定义，不再重复展开整块读键逻辑。
  3. 当前块只处理“读键”，不负责编码灯输出。
*)
FUNCTION_BLOCK FB_PanelReader
VAR_IN_OUT
    stPanelButtons: ST_PanelButtons;     // 综合面板按键结构；调用方先写入真实输入映射，本块再统一回写全部逻辑键值。
END_VAR
VAR_INPUT
    uiIN0: UINT;                         // 面板输入字 0；承载当前型号的真实物理输入位。
    uiIN1: UINT;                         // 面板输入字 1；承载当前型号的真实物理输入位。
    uiIN2: UINT;                         // 面板输入字 2；承载当前型号的真实物理输入位。
    uiIN3: UINT;                         // 面板输入字 3；承载当前型号的真实物理输入位。
END_VAR

stPanelButtons.stManual.bValue := F_PanelReadKeyByOrder(uiInputWordIndex := stPanelButtons.stManual.uiInputWordIndex, uiInputBitIndex := stPanelButtons.stManual.uiInputBitIndex, uiIN0 := uiIN0, uiIN1 := uiIN1, uiIN2 := uiIN2, uiIN3 := uiIN3);                         // 读取手动键当前值。
stPanelButtons.stSemiautomatic.bValue := F_PanelReadKeyByOrder(uiInputWordIndex := stPanelButtons.stSemiautomatic.uiInputWordIndex, uiInputBitIndex := stPanelButtons.stSemiautomatic.uiInputBitIndex, uiIN0 := uiIN0, uiIN1 := uiIN1, uiIN2 := uiIN2, uiIN3 := uiIN3);          // 读取半自动键当前值。
stPanelButtons.stAutomatic.bValue := F_PanelReadKeyByOrder(uiInputWordIndex := stPanelButtons.stAutomatic.uiInputWordIndex, uiInputBitIndex := stPanelButtons.stAutomatic.uiInputBitIndex, uiIN0 := uiIN0, uiIN1 := uiIN1, uiIN2 := uiIN2, uiIN3 := uiIN3);                  // 读取全自动键当前值。
stPanelButtons.stAdjustMold.bValue := F_PanelReadKeyByOrder(uiInputWordIndex := stPanelButtons.stAdjustMold.uiInputWordIndex, uiInputBitIndex := stPanelButtons.stAdjustMold.uiInputBitIndex, uiIN0 := uiIN0, uiIN1 := uiIN1, uiIN2 := uiIN2, uiIN3 := uiIN3);                // 读取调模键当前值。
stPanelButtons.stHeat.bValue := F_PanelReadKeyByOrder(uiInputWordIndex := stPanelButtons.stHeat.uiInputWordIndex, uiInputBitIndex := stPanelButtons.stHeat.uiInputBitIndex, uiIN0 := uiIN0, uiIN1 := uiIN1, uiIN2 := uiIN2, uiIN3 := uiIN3);                               // 读取电热键当前值。
stPanelButtons.stMotor.bValue := F_PanelReadKeyByOrder(uiInputWordIndex := stPanelButtons.stMotor.uiInputWordIndex, uiInputBitIndex := stPanelButtons.stMotor.uiInputBitIndex, uiIN0 := uiIN0, uiIN1 := uiIN1, uiIN2 := uiIN2, uiIN3 := uiIN3);                            // 读取马达键当前值。
stPanelButtons.stMoldOpen.bValue := F_PanelReadKeyByOrder(uiInputWordIndex := stPanelButtons.stMoldOpen.uiInputWordIndex, uiInputBitIndex := stPanelButtons.stMoldOpen.uiInputBitIndex, uiIN0 := uiIN0, uiIN1 := uiIN1, uiIN2 := uiIN2, uiIN3 := uiIN3);                      // 读取开模键当前值。
stPanelButtons.stMoldClose.bValue := F_PanelReadKeyByOrder(uiInputWordIndex := stPanelButtons.stMoldClose.uiInputWordIndex, uiInputBitIndex := stPanelButtons.stMoldClose.uiInputBitIndex, uiIN0 := uiIN0, uiIN1 := uiIN1, uiIN2 := uiIN2, uiIN3 := uiIN3);                    // 读取锁模键当前值。
stPanelButtons.stMaterialMelt.bValue := F_PanelReadKeyByOrder(uiInputWordIndex := stPanelButtons.stMaterialMelt.uiInputWordIndex, uiInputBitIndex := stPanelButtons.stMaterialMelt.uiInputBitIndex, uiIN0 := uiIN0, uiIN1 := uiIN1, uiIN2 := uiIN2, uiIN3 := uiIN3);              // 读取储料键当前值。
stPanelButtons.stCleanMaterial.bValue := F_PanelReadKeyByOrder(uiInputWordIndex := stPanelButtons.stCleanMaterial.uiInputWordIndex, uiInputBitIndex := stPanelButtons.stCleanMaterial.uiInputBitIndex, uiIN0 := uiIN0, uiIN1 := uiIN1, uiIN2 := uiIN2, uiIN3 := uiIN3);            // 读取清料键当前值。
stPanelButtons.stJetLube.bValue := F_PanelReadKeyByOrder(uiInputWordIndex := stPanelButtons.stJetLube.uiInputWordIndex, uiInputBitIndex := stPanelButtons.stJetLube.uiInputBitIndex, uiIN0 := uiIN0, uiIN1 := uiIN1, uiIN2 := uiIN2, uiIN3 := uiIN3);                         // 读取润滑键当前值。
stPanelButtons.stInjFwd.bValue := F_PanelReadKeyByOrder(uiInputWordIndex := stPanelButtons.stInjFwd.uiInputWordIndex, uiInputBitIndex := stPanelButtons.stInjFwd.uiInputBitIndex, uiIN0 := uiIN0, uiIN1 := uiIN1, uiIN2 := uiIN2, uiIN3 := uiIN3);                           // 读取射出键当前值。
stPanelButtons.stInjBwd.bValue := F_PanelReadKeyByOrder(uiInputWordIndex := stPanelButtons.stInjBwd.uiInputWordIndex, uiInputBitIndex := stPanelButtons.stInjBwd.uiInputBitIndex, uiIN0 := uiIN0, uiIN1 := uiIN1, uiIN2 := uiIN2, uiIN3 := uiIN3);                           // 读取射退键当前值。
stPanelButtons.stPressRise.bValue := F_PanelReadKeyByOrder(uiInputWordIndex := stPanelButtons.stPressRise.uiInputWordIndex, uiInputBitIndex := stPanelButtons.stPressRise.uiInputBitIndex, uiIN0 := uiIN0, uiIN1 := uiIN1, uiIN2 := uiIN2, uiIN3 := uiIN3);                      // 读取压力加键当前值。
stPanelButtons.stPressFall.bValue := F_PanelReadKeyByOrder(uiInputWordIndex := stPanelButtons.stPressFall.uiInputWordIndex, uiInputBitIndex := stPanelButtons.stPressFall.uiInputBitIndex, uiIN0 := uiIN0, uiIN1 := uiIN1, uiIN2 := uiIN2, uiIN3 := uiIN3);                      // 读取压力减键当前值。
stPanelButtons.stEjectorFwd.bValue := F_PanelReadKeyByOrder(uiInputWordIndex := stPanelButtons.stEjectorFwd.uiInputWordIndex, uiInputBitIndex := stPanelButtons.stEjectorFwd.uiInputBitIndex, uiIN0 := uiIN0, uiIN1 := uiIN1, uiIN2 := uiIN2, uiIN3 := uiIN3);                    // 读取托模进键当前值。
stPanelButtons.stEjectorBwd.bValue := F_PanelReadKeyByOrder(uiInputWordIndex := stPanelButtons.stEjectorBwd.uiInputWordIndex, uiInputBitIndex := stPanelButtons.stEjectorBwd.uiInputBitIndex, uiIN0 := uiIN0, uiIN1 := uiIN1, uiIN2 := uiIN2, uiIN3 := uiIN3);                    // 读取托模退键当前值。
stPanelButtons.stMultiEjector.bValue := F_PanelReadKeyByOrder(uiInputWordIndex := stPanelButtons.stMultiEjector.uiInputWordIndex, uiInputBitIndex := stPanelButtons.stMultiEjector.uiInputBitIndex, uiIN0 := uiIN0, uiIN1 := uiIN1, uiIN2 := uiIN2, uiIN3 := uiIN3);                // 读取多次托模键当前值。
stPanelButtons.stBlow.bValue := F_PanelReadKeyByOrder(uiInputWordIndex := stPanelButtons.stBlow.uiInputWordIndex, uiInputBitIndex := stPanelButtons.stBlow.uiInputBitIndex, uiIN0 := uiIN0, uiIN1 := uiIN1, uiIN2 := uiIN2, uiIN3 := uiIN3);                               // 读取吹气键当前值。
stPanelButtons.stInjUnitFwd.bValue := F_PanelReadKeyByOrder(uiInputWordIndex := stPanelButtons.stInjUnitFwd.uiInputWordIndex, uiInputBitIndex := stPanelButtons.stInjUnitFwd.uiInputBitIndex, uiIN0 := uiIN0, uiIN1 := uiIN1, uiIN2 := uiIN2, uiIN3 := uiIN3);                    // 读取座进键当前值。
stPanelButtons.stInjUnitBwd.bValue := F_PanelReadKeyByOrder(uiInputWordIndex := stPanelButtons.stInjUnitBwd.uiInputWordIndex, uiInputBitIndex := stPanelButtons.stInjUnitBwd.uiInputBitIndex, uiIN0 := uiIN0, uiIN1 := uiIN1, uiIN2 := uiIN2, uiIN3 := uiIN3);                    // 读取座退键当前值。
stPanelButtons.stLockFwd.bValue := F_PanelReadKeyByOrder(uiInputWordIndex := stPanelButtons.stLockFwd.uiInputWordIndex, uiInputBitIndex := stPanelButtons.stLockFwd.uiInputBitIndex, uiIN0 := uiIN0, uiIN1 := uiIN1, uiIN2 := uiIN2, uiIN3 := uiIN3);                          // 读取定位进键当前值。
stPanelButtons.stLockBwd.bValue := F_PanelReadKeyByOrder(uiInputWordIndex := stPanelButtons.stLockBwd.uiInputWordIndex, uiInputBitIndex := stPanelButtons.stLockBwd.uiInputBitIndex, uiIN0 := uiIN0, uiIN1 := uiIN1, uiIN2 := uiIN2, uiIN3 := uiIN3);                          // 读取定位退键当前值。
stPanelButtons.stCoreFwdA.bValue := F_PanelReadKeyByOrder(uiInputWordIndex := stPanelButtons.stCoreFwdA.uiInputWordIndex, uiInputBitIndex := stPanelButtons.stCoreFwdA.uiInputBitIndex, uiIN0 := uiIN0, uiIN1 := uiIN1, uiIN2 := uiIN2, uiIN3 := uiIN3);                        // 读取中子 A 进键当前值。
stPanelButtons.stCoreBwdA.bValue := F_PanelReadKeyByOrder(uiInputWordIndex := stPanelButtons.stCoreBwdA.uiInputWordIndex, uiInputBitIndex := stPanelButtons.stCoreBwdA.uiInputBitIndex, uiIN0 := uiIN0, uiIN1 := uiIN1, uiIN2 := uiIN2, uiIN3 := uiIN3);                        // 读取中子 A 退键当前值。
stPanelButtons.stZipperBwd.bValue := F_PanelReadKeyByOrder(uiInputWordIndex := stPanelButtons.stZipperBwd.uiInputWordIndex, uiInputBitIndex := stPanelButtons.stZipperBwd.uiInputBitIndex, uiIN0 := uiIN0, uiIN1 := uiIN1, uiIN2 := uiIN2, uiIN3 := uiIN3);                      // 读取倒带键当前值。
stPanelButtons.stZipperFwd.bValue := F_PanelReadKeyByOrder(uiInputWordIndex := stPanelButtons.stZipperFwd.uiInputWordIndex, uiInputBitIndex := stPanelButtons.stZipperFwd.uiInputBitIndex, uiIN0 := uiIN0, uiIN1 := uiIN1, uiIN2 := uiIN2, uiIN3 := uiIN3);                      // 读取拉带键当前值。
stPanelButtons.stZipperClamp.bValue := F_PanelReadKeyByOrder(uiInputWordIndex := stPanelButtons.stZipperClamp.uiInputWordIndex, uiInputBitIndex := stPanelButtons.stZipperClamp.uiInputBitIndex, uiIN0 := uiIN0, uiIN1 := uiIN1, uiIN2 := uiIN2, uiIN3 := uiIN3);                  // 读取夹带键当前值。
stPanelButtons.stZipperMotor.bValue := F_PanelReadKeyByOrder(uiInputWordIndex := stPanelButtons.stZipperMotor.uiInputWordIndex, uiInputBitIndex := stPanelButtons.stZipperMotor.uiInputBitIndex, uiIN0 := uiIN0, uiIN1 := uiIN1, uiIN2 := uiIN2, uiIN3 := uiIN3);                  // 读取拉带马达键当前值。
END_FUNCTION_BLOCK
